# EPICS substitutions: fastFeedbackApp/Db/common/bsaATTR.substitutions
#==============================================================================
#
# Abs:  Beam Synchronous Acquisition records for a single Toroid.
#
# Name: bsaATTR.substitutions
#
# Note: Must follow the LCLS naming conventions.
#
#==============================================================================
# BSA Integration Note:
# Each device attribute (such as width ) provides input to bsaEdefAvg.db.
# The bsaEdefAvg.db provides the RMS and Avg -$(DEV):$(SECN)<edef id>, and history -
#   $(DEV):$(SECN)HST<edef id> for each device attribute for each of 20 edefs.
#
file bsaATTREdef.db
{
#	      Device   Name                                                      Init
#                                                                                Event Code
  pattern {D ,  ATTR ,  I  ,  EG  ,  HO  ,  LO  ,PR,  AD  , SINK_SIZE       , }
	   { $(D),  S1BSA, $(I), $(EG), $(HO), $(LO), 3, $(AD), $(SINK_SIZE\=10) }
	   { $(D),  S2BSA, $(I), $(EG), $(HO), $(LO), 3, $(AD), $(SINK_SIZE\=10) }
  	   { $(D),  S3BSA, $(I), $(EG), $(HO), $(LO), 3, $(AD), $(SINK_SIZE\=10) }
       { $(D),  S4BSA, $(I), $(EG), $(HO), $(LO), 3, $(AD), $(SINK_SIZE\=10) }
	   { $(D),  S5BSA, $(I), $(EG), $(HO), $(LO), 3, $(AD), $(SINK_SIZE\=10) }
	   { $(D),  S6BSA, $(I), $(EG), $(HO), $(LO), 3, $(AD), $(SINK_SIZE\=10) }
	   { $(D),  S7BSA, $(I), $(EG), $(HO), $(LO), 3, $(AD), $(SINK_SIZE\=10) }
	   { $(D),  S8BSA, $(I), $(EG), $(HO), $(LO), 3, $(AD), $(SINK_SIZE\=10) }
	   { $(D),  S9BSA, $(I), $(EG), $(HO), $(LO), 3, $(AD), $(SINK_SIZE\=10) }
	   { $(D), S10BSA, $(I), $(EG), $(HO), $(LO), 3, $(AD), $(SINK_SIZE\=10) }
}

file bsaEdefFanouts.db
{
#	    Device  Name
  pattern {  DEV ,  SECN , INP , EGU  ,HOPR ,LOPR ,PREC ,ADEL ,FLNK   }
	  { $(D) ,$(ATTR), $(I),$(EG) ,$(HO),$(LO),$(PR),$(AD),$(LNK) }
}
